// Mitsubishi GX Works2 project: 0630실린더 응용동작 3코멘트   PLC: Q02/Q02H

PROGRAM MAIN
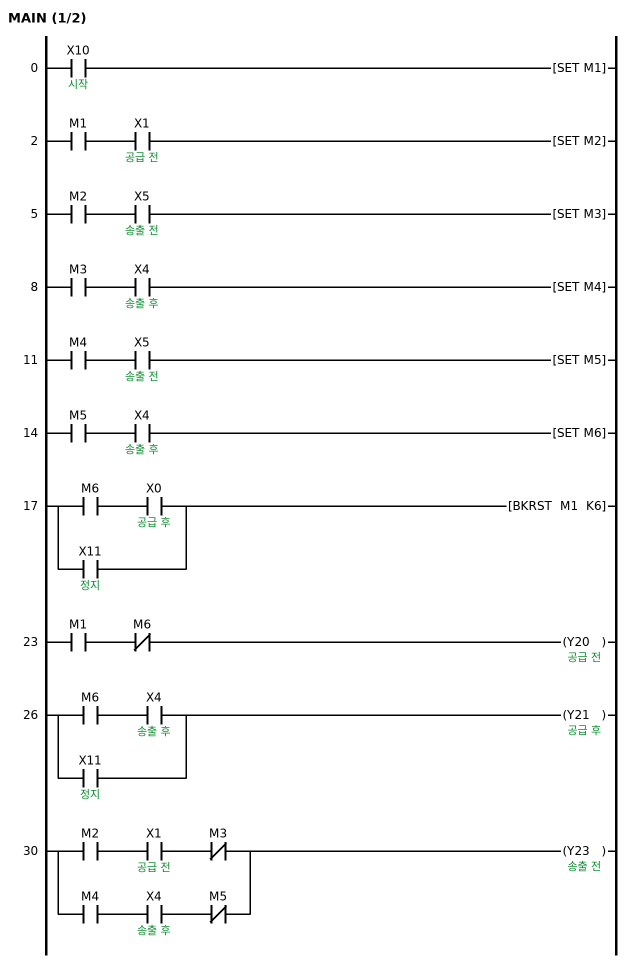
0     LD      X10  ; 시작
      SET     M1
2     LD      M1
      AND     X1  ; 공급 전
      SET     M2
5     LD      M2
      AND     X5  ; 송출 전
      SET     M3
8     LD      M3
      AND     X4  ; 송출 후
      SET     M4
11    LD      M4
      AND     X5  ; 송출 전
      SET     M5
14    LD      M5
      AND     X4  ; 송출 후
      SET     M6
17    LD      M6
      AND     X0  ; 공급 후
      OR      X11  ; 정지
      BKRST   M1 K6
23    LD      M1
      ANI     M6
      OUT     Y20  ; 공급 전
26    LD      M6
      AND     X4  ; 송출 후
      OR      X11  ; 정지
      OUT     Y21  ; 공급 후
30    LD      M2
      AND     X1  ; 공급 전
      ANI     M3
      LD      M4
      AND     X4  ; 송출 후
      ANI     M5
      ORB
      OUT     Y23  ; 송출 전
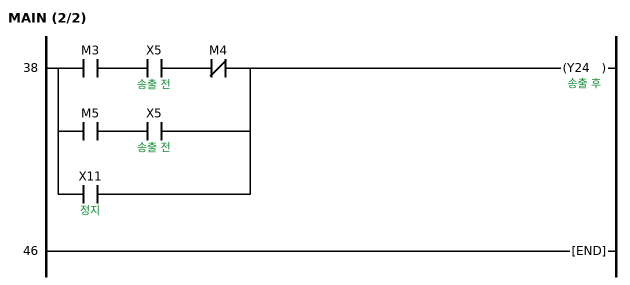
38    LD      M3
      AND     X5  ; 송출 전
      ANI     M4
      LD      M5
      AND     X5  ; 송출 전
      ORB
      OR      X11  ; 정지
      OUT     Y24  ; 송출 후
46    END
END_PROGRAM

// device comments not shown above
X2  ; 드릴 상
X3  ; 드릴 하
X6  ; 배출 후
X7  ; 배출 전
Y22  ; 드릴 전
Y25  ; 배출 전
Y26  ; 배출 후
